// TwinCAT 3 PLC project Demo
// ProgramVersion: 3.1.4024.0
// libraries:
//   Tc2_Standard, * (Beckhoff Automation GmbH)
// project tree:
//   DUTs/ E_Mode.TcDUT, ST_Sample.TcDUT
//   GVLs/ GVL_Main.TcGVL
//   POUs/ I_Counter.TcIO, FB_Counter.TcPOU, PRG_Stats.TcPOU, MAIN.TcPOU
//   POUs/Drafts/ FB_Draft.TcPOU
//   / PlcTask.TcTTO
//   Visu/ Visualization.TcVIS (not stored)

CONFIGURATION Demo
    RESOURCE PLC ON TwinCAT3
        TASK PlcTask(INTERVAL := T#10ms, PRIORITY := 20);
        PROGRAM MAIN WITH PlcTask : MAIN;
    END_RESOURCE
END_CONFIGURATION

// ---- DUTs/E_Mode.TcDUT
{attribute 'qualified_only'}
{attribute 'strict'}
TYPE E_Mode :
(
    Idle := 0,
    Running := 10,
    Done
) INT;
END_TYPE

// ---- DUTs/ST_Sample.TcDUT
TYPE ST_Sample :
STRUCT
    nValue : DINT;
    fScale : LREAL := 2.5;
    eMode  : E_Mode := E_Mode.Idle;
    aLast  : ARRAY[1..GVL_Main.MAX_STEP] OF DINT;
END_STRUCT
END_TYPE

// ---- GVLs/GVL_Main.TcGVL
{attribute 'qualified_only'}
VAR_GLOBAL
    nScans : UDINT;
    bTimerDone : BOOL;
END_VAR
VAR_GLOBAL CONSTANT
    MAX_STEP : DINT := 7;
END_VAR

// ---- POUs/I_Counter.TcIO
INTERFACE I_Counter

METHOD Increment : BOOL
END_METHOD

PROPERTY Step : DINT
GET
END_GET
SET
END_SET
END_PROPERTY

END_INTERFACE

// ---- POUs/MAIN.TcPOU
PROGRAM MAIN
VAR
    fbCounter : FB_Counter;
    itfCounter : I_Counter;
    fbTimer : Tc2_Standard.TON;
    fbEdge : R_TRIG;
    stSample : ST_Sample;
    eMode : E_Mode := E_Mode.Idle;
    nStepSeen : DINT;
    bAtLimit : BOOL;
    bLimitReached : BOOL;
    bTimerQ : BOOL;
    nItfStep : DINT;
    nStatsMax : DINT;
    nStatsMean : DINT;
    nLast : DINT;
    // A POU constant, read through the POU's name.
    aHistory : ARRAY[1..FB_Counter.HISTORY_LEN] OF DINT;
    nHistoryLen : INT;
    nHistoryLast : DINT;
END_VAR

// Scan counter in a qualified-only GVL.
GVL_Main.nScans := GVL_Main.nScans + 1;

// Property write and read, method call, action call.
IF GVL_Main.nScans = 1 THEN
    fbCounter.Step := GVL_Main.MAX_STEP;
    itfCounter := fbCounter;
END_IF
nStepSeen := fbCounter.Step;
fbCounter(bEnable := TRUE);
bAtLimit := fbCounter.AtLimit;
bLimitReached S= bAtLimit AND_THEN fbCounter.nCount >= 100;
IF fbCounter.nCount >= 100 THEN
    fbCounter.Reset();
END_IF

// Interface property access.
nItfStep := itfCounter.Step;

// A Tc2_Standard timer and edge detection.
fbTimer(IN := TRUE, PT := T#50MS);
fbEdge(CLK := fbTimer.Q);
bTimerQ := fbTimer.Q;
IF fbEdge.Q THEN
    GVL_Main.bTimerDone := TRUE;
END_IF

// Another PROGRAM, not in any task: it runs when MAIN calls it. Its
// method, property and action are reached through its name.
PRG_Stats(nSample := fbCounter.nCount);
nStatsMax := PRG_Stats.nMax;
nStatsMean := PRG_Stats.Mean;
IF fbCounter.nCount = 0 THEN
    PRG_Stats.Clear();
END_IF

// DUT struct and enum.
stSample.nValue := stSample.nValue + 1;
stSample.aLast[GVL_Main.MAX_STEP] := stSample.nValue * 100;
nLast := stSample.aLast[7];
CASE eMode OF
    E_Mode.Idle: eMode := E_Mode.Running;
    E_Mode.Running: IF stSample.nValue >= 3 THEN eMode := E_Mode.Done; END_IF
END_CASE

nHistoryLen := FB_Counter.HISTORY_LEN;
aHistory[FB_Counter.HISTORY_LEN] := fbCounter.nCount;
nHistoryLast := aHistory[4];

END_PROGRAM

// ---- POUs/FB_Counter.TcPOU
{attribute 'reflection'}
FUNCTION_BLOCK FB_Counter IMPLEMENTS I_Counter
VAR_INPUT
    bEnable : BOOL;
END_VAR
VAR_OUTPUT
    nCount : DINT;
END_VAR
VAR
    nStep : DINT := 1;
    nLimit : DINT := 100;
    nResets : INT;
END_VAR
VAR CONSTANT
    HISTORY_LEN : INT := 4;
END_VAR

IF bEnable THEN
    Increment();
END_IF

METHOD PUBLIC Increment : BOOL
VAR
    nNext : DINT;
END_VAR
nNext := nCount + nStep;
IF nNext > nLimit THEN
    nNext := nLimit;
END_IF
nCount := nNext;
Increment := nCount = nLimit;
END_METHOD

PROPERTY PUBLIC Step : DINT
GET
Step := nStep;
END_GET
SET
IF Step > 0 THEN
    nStep := Step;
END_IF
END_SET
END_PROPERTY

PROPERTY AtLimit : BOOL
GET
AtLimit := nCount >= nLimit;
END_GET
END_PROPERTY

ACTION Reset:
nCount := 0;
nResets := nResets + 1;
END_ACTION

END_FUNCTION_BLOCK

// ---- POUs/PRG_Stats.TcPOU
PROGRAM PRG_Stats
VAR_INPUT
    nSample : DINT;
END_VAR
VAR_OUTPUT
    nMax : DINT;
END_VAR
VAR
    nCalls : UDINT;
    nSum : DINT;
END_VAR

nCalls := nCalls + 1;
Accumulate(nSample);

METHOD PRIVATE Accumulate
VAR_INPUT
    nValue : DINT;
END_VAR
nSum := nSum + nValue;
IF nValue > nMax THEN
    nMax := nValue;
END_IF
END_METHOD

PROPERTY Mean : DINT
GET
IF nCalls > 0 THEN
    Mean := nSum / UDINT_TO_DINT(nCalls);
END_IF
END_GET
END_PROPERTY

ACTION Clear:
nCalls := 0;
nSum := 0;
nMax := 0;
END_ACTION

END_PROGRAM

// ---- POUs/Drafts/FB_Draft.TcPOU
// Unfinished, and excluded from the build (the POUs\Drafts folder has
// ExcludeFromBuild): the project compiles without it.
FUNCTION_BLOCK FB_Draft
VAR
    nValue : DINT;
END_VAR

nValue :=

END_FUNCTION_BLOCK
